// TIA Portal V17 export
// export: Created 2021-09-22T11:16:29.8821443Z, ExportSetting WithDefaults, DisplayName Totally Integrated Automation Portal, DisplayVersion V17, DisplayName TIA Portal Openness, DisplayVersion V17, DisplayName TIA Portal Version Control Interface, DisplayVersion V17, DisplayName SINAMICS Startdrive Advanced, DisplayVersion V17, DisplayName SINAMICS Startdrive G130, G150, S120, S150, SINAMICS MV, S210, DisplayVersion V17, DisplayName SINAMICS Startdrive G110M, G120, G120C, G120D, G120P, G115D, DisplayVersion V17, DisplayName STEP 7 Professional, DisplayVersion V17, DisplayName STEP 7 Safety, DisplayVersion V17, DisplayName WinCC Advanced / Unified PC, DisplayVersion V17
VAR_GLOBAL   // PLC tag table "SystemConstant"
END_VAR
VAR_GLOBAL CONSTANT   // user constants
   ERR_FUB_NOT_ENABLED : UInt := 65534;
   ERR_BUSY : UInt := 65535;
   ERR_FUB_INPUT_PARAMETER : UInt := 62000;
   ERR_OK : UInt := 0;
   ERR_UNDEFINED : UInt := 65533;
   ERR_SAFETY_NOK : UInt := 65531;
   ERR_FUB_ERROR : UInt := 65530;
   ERR_BARRIER_NOK : UInt := 65532;
   ERR_AIR_NOK : UInt := 65529;
END_VAR
